Staubli VAL3: mergeList.pgx

public program mergeList()
begin
end
